// Mitsubishi GX Works2 project: Control3Light   PLC: FX3U/FX3UC

PROGRAM MAIN
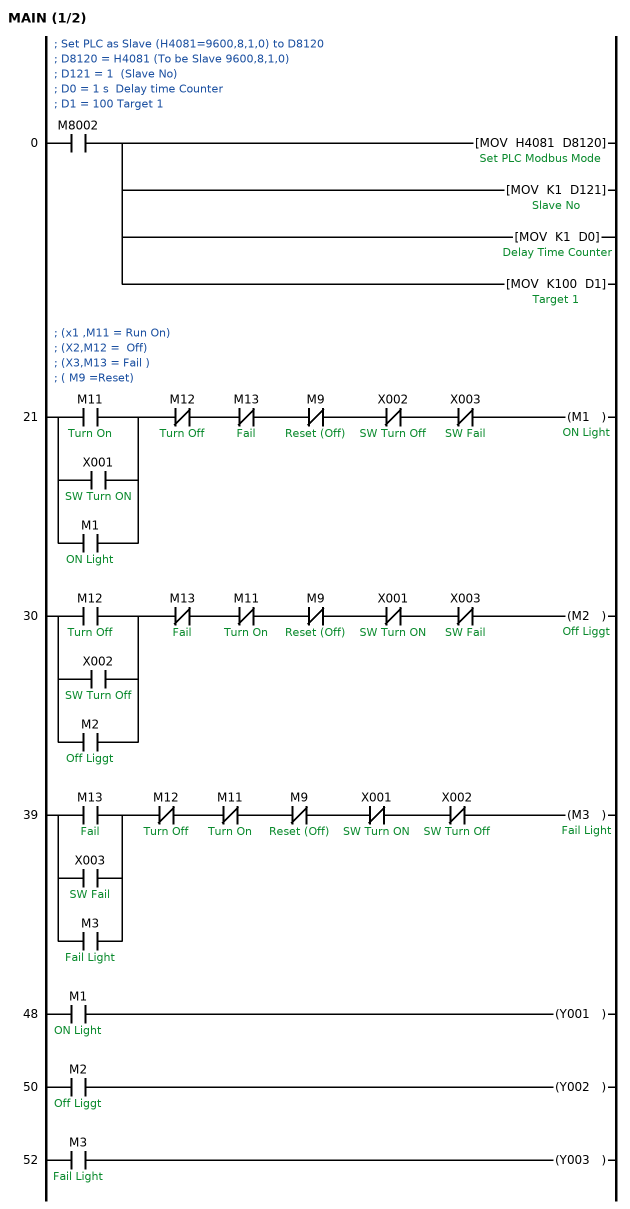
; Set PLC as Slave (H4081=9600,8,1,0) to D8120
; D8120 = H4081 (To be Slave 9600,8,1,0)
; D121 = 1  (Slave No)
; D0 = 1 s  Delay time Counter
; D1 = 100 Target 1
0     LD      M8002
      MOV     H4081 D8120  ; Set PLC Modbus Mode
      MOV     K1 D121  ; Slave No
      MOV     K1 D0  ; Delay Time Counter
      MOV     K100 D1  ; Target 1
; (x1 ,M11 = Run On)
; (X2,M12 =  Off)
; (X3,M13 = Fail )
; ( M9 =Reset)
21    LD      M11  ; Turn On
      OR      X001  ; SW Turn ON
      OR      M1  ; ON Light
      ANI     M12  ; Turn Off
      ANI     M13  ; Fail
      ANI     M9  ; Reset (Off)
      ANI     X002  ; SW Turn Off
      ANI     X003  ; SW Fail
      OUT     M1  ; ON Light
30    LD      M12  ; Turn Off
      OR      X002  ; SW Turn Off
      OR      M2  ; Off Liggt
      ANI     M13  ; Fail
      ANI     M11  ; Turn On
      ANI     M9  ; Reset (Off)
      ANI     X001  ; SW Turn ON
      ANI     X003  ; SW Fail
      OUT     M2  ; Off Liggt
39    LD      M13  ; Fail
      OR      X003  ; SW Fail
      OR      M3  ; Fail Light
      ANI     M12  ; Turn Off
      ANI     M11  ; Turn On
      ANI     M9  ; Reset (Off)
      ANI     X001  ; SW Turn ON
      ANI     X002  ; SW Turn Off
      OUT     M3  ; Fail Light
48    LD      M1  ; ON Light
      OUT     Y001
50    LD      M2  ; Off Liggt
      OUT     Y002
52    LD      M3  ; Fail Light
      OUT     Y003
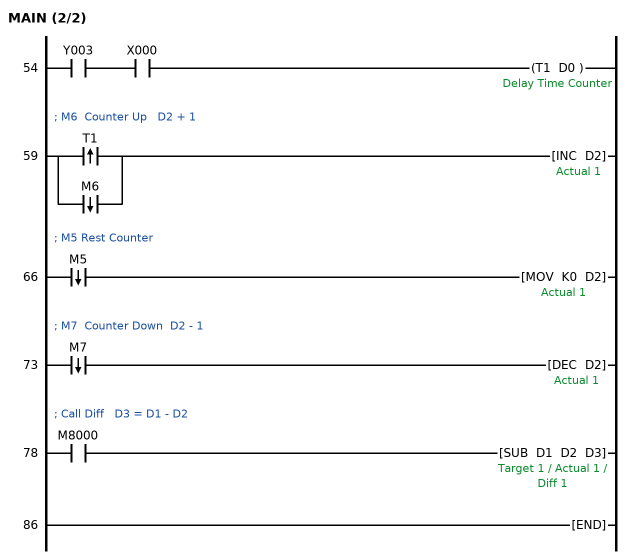
54    LD      Y003
      AND     X000
      OUT     T1 D0  ; Delay Time Counter
; M6  Counter Up   D2 + 1
59    LDP     T1
      ORF     M6
      INC     D2  ; Actual 1
; M5 Rest Counter
66    LDF     M5
      MOV     K0 D2
; M7  Counter Down  D2 - 1
73    LDF     M7
      DEC     D2
; Call Diff   D3 = D1 - D2
78    LD      M8000
      SUB     D1 D2 D3  ; Diff 1
86    END
END_PROGRAM
